{attribute 'qualified_only'}
VAR_GLOBAL PERSISTENT
	// PID variables are stored so the tuner does not have to run each time
	kp: REAL := 0.196;
	ki: REAL := 0.00326;
	kd: REAL := 0;
END_VAR

VAR_GLOBAL
	iHeaterActuator: INT := 0;	// Heater power (0-100%)
	rSetpoint: REAL := 35.0;	// Target temperature (°C)
	
	rTempSensor: REAL := 0.0;	// Temperature (°C)
	iRealPower: INT := 0;		// Actual heater power (W)
	
	doTuning: BOOL := FALSE; 	// Whether or not to run the tuner
END_VAR

(* stored: Version 1.1.0.1, ProductVersion 3.1.4024.12
   GVL GVL: Id {55000c09-fd3e-4ef2-bc8e-0182699637fa} *)
